(* IEC 61131-3 sources: ISN2023_SystSecurity/TP/fichers linux/sec_sys_auto01_12/PLC_project_deux/build, 2 files *)

(* ---- plc.st ---- *)
TYPE
  LOGLEVEL : (CRITICAL, WARNING, INFO, DEBUG) := INFO;
END_TYPE

FUNCTION_BLOCK LOGGER
  VAR_INPUT
    TRIG : BOOL;
    MSG : STRING;
    LEVEL : LOGLEVEL := INFO;
  END_VAR
  VAR
    TRIG0 : BOOL;
  END_VAR

  IF TRIG AND NOT TRIG0 THEN
  {{
   LogMessage(GetFbVar(LEVEL),(char*)GetFbVar(MSG, .body),GetFbVar(MSG, .len));
  }}
  END_IF;
  TRIG0:=TRIG;
END_FUNCTION_BLOCK

FUNCTION_BLOCK python_eval
  VAR_INPUT
    TRIG : BOOL;
    CODE : STRING;
  END_VAR
  VAR_OUTPUT
    ACK : BOOL;
    RESULT : STRING;
  END_VAR
  VAR
    STATE : DWORD;
    BUFFER : STRING;
    PREBUFFER : STRING;
    TRIGM1 : BOOL;
    TRIGGED : BOOL;
  END_VAR

  {extern void __PythonEvalFB(int, PYTHON_EVAL*);__PythonEvalFB(0, data__);}
END_FUNCTION_BLOCK

FUNCTION_BLOCK python_poll
  VAR_INPUT
    TRIG : BOOL;
    CODE : STRING;
  END_VAR
  VAR_OUTPUT
    ACK : BOOL;
    RESULT : STRING;
  END_VAR
  VAR
    STATE : DWORD;
    BUFFER : STRING;
    PREBUFFER : STRING;
    TRIGM1 : BOOL;
    TRIGGED : BOOL;
  END_VAR

  {extern void __PythonEvalFB(int, PYTHON_EVAL*);__PythonEvalFB(1,(PYTHON_EVAL*)(void*)data__);}
END_FUNCTION_BLOCK

FUNCTION_BLOCK python_gear
  VAR_INPUT
    N : UINT;
    TRIG : BOOL;
    CODE : STRING;
  END_VAR
  VAR_OUTPUT
    ACK : BOOL;
    RESULT : STRING;
  END_VAR
  VAR
    py_eval : python_eval;
    COUNTER : UINT;
    _TMP_ADD10_OUT : UINT;
    _TMP_EQ13_OUT : BOOL;
    _TMP_SEL15_OUT : UINT;
    _TMP_AND7_OUT : BOOL;
  END_VAR

  _TMP_ADD10_OUT := ADD(COUNTER, 1);
  _TMP_EQ13_OUT := EQ(N, _TMP_ADD10_OUT);
  _TMP_SEL15_OUT := SEL(_TMP_EQ13_OUT, _TMP_ADD10_OUT, 0);
  COUNTER := _TMP_SEL15_OUT;
  _TMP_AND7_OUT := AND(_TMP_EQ13_OUT, TRIG);
  py_eval(TRIG := _TMP_AND7_OUT, CODE := CODE);
  ACK := py_eval.ACK;
  RESULT := py_eval.RESULT;
END_FUNCTION_BLOCK

PROGRAM program2
  VAR
    START_BUTTON : BOOL := 0;
    LEVEL_SENSOR : BOOL := 0;
    CONTACT_SENSOR : BOOL := 0;
    MOTOR : BOOL := 0;
    NOZZLE : BOOL := 0;
    RUN : BOOL := 0;
  END_VAR

  RUN := START_BUTTON;
  MOTOR := (LEVEL_SENSOR OR NOT(CONTACT_SENSOR)) AND RUN;
  IF NOT(CONTACT_SENSOR) AND RUN AND LEVEL_SENSOR AND RUN THEN
    NOZZLE := FALSE; (*reset*)
  END_IF;
  NOZZLE := NOT(LEVEL_SENSOR) AND CONTACT_SENSOR AND RUN;
  IF NOT(LEVEL_SENSOR) AND CONTACT_SENSOR AND RUN THEN
    MOTOR := FALSE; (*reset*)
  END_IF;
END_PROGRAM

CONFIGURATION Config0

  RESOURCE Res0 ON PLC
    TASK task0(INTERVAL := T#20ms,PRIORITY := 0);
    PROGRAM instance0 WITH task0 : program2;
  END_RESOURCE
END_CONFIGURATION

(* ---- generated_plc.st ---- *)
PROGRAM program2
  VAR
    START_BUTTON AT %QX0.0 : BOOL := 0;
    LEVEL_SENSOR AT %QX0.1 : BOOL := 0;
    CONTACT_SENSOR AT %QX0.2 : BOOL := 0;
    MOTOR AT %QX0.3 : BOOL := 0;
    NOZZLE AT %QX0.4 : BOOL := 0;
    RUN AT %QX0.5 : BOOL := 0;
  END_VAR

  RUN := START_BUTTON;
  MOTOR := (LEVEL_SENSOR OR NOT(CONTACT_SENSOR)) AND RUN;
  IF NOT(CONTACT_SENSOR) AND RUN AND LEVEL_SENSOR AND RUN THEN
    NOZZLE := FALSE; (*reset*)
  END_IF;
  NOZZLE := NOT(LEVEL_SENSOR) AND CONTACT_SENSOR AND RUN;
  IF NOT(LEVEL_SENSOR) AND CONTACT_SENSOR AND RUN THEN
    MOTOR := FALSE; (*reset*)
  END_IF;
END_PROGRAM

CONFIGURATION Config0

  RESOURCE Res0 ON PLC
    TASK task0(INTERVAL := T#20ms,PRIORITY := 0);
    PROGRAM instance0 WITH task0 : program2;
  END_RESOURCE
END_CONFIGURATION
